FUNCTION_BLOCK AX_RangeBasedPulse (* Generates a pulse on AX adapter based on distance traveled (Adapter Version) *)
  (* Standard: 61499-2; Description: Copyright (c) 2026 HR Agrartechnik GmbH This program and the accompanying materials are made available under the terms of the Eclipse Public License 2.0 which is available at https://www.eclipse.org/legal/epl-2.0/ SPDX-License-Identifier: EPL-2.0 *)
  (* Version 1.0, 2026-04-19, Franz Höpfinger, HR Agrartechnik GmbH, initial API and implementation *)
  PACKAGE logiBUS::signalprocessing::distance;
  IMPORT eclipse4diac::core::TypeHash;
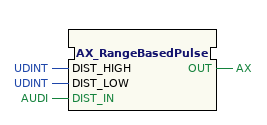
  VAR_INPUT
    DIST_HIGH : UDINT := 5000; (* Distance for HIGH pulse (mm) *)
    DIST_LOW : UDINT := 5000; (* Distance for LOW pulse (mm) *)
  END_VAR
  SOCKETS
    DIST_IN : adapter::types::unidirectional::AUDI; (* Input Distance Adapter *)
  END_SOCKETS
  PLUGS
    OUT : adapter::types::unidirectional::AX; (* Pulse Output Adapter *)
  END_PLUGS
  VAR
    LastDist : UDINT; (* Last distance value when state changed *)
    FirstRun : BOOL := TRUE; (* Initial run flag *)
    LastState : BOOL; (* Last state of Q *)
  END_VAR
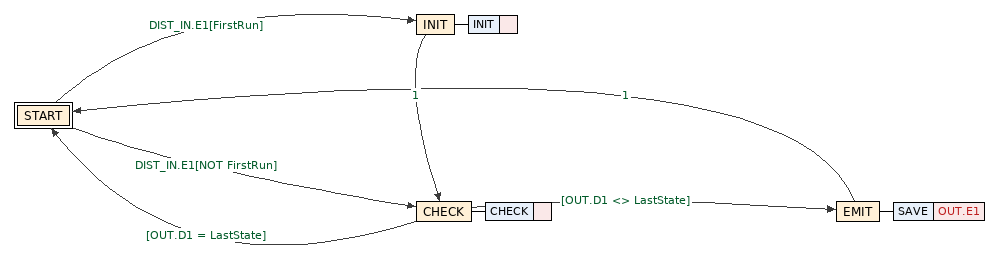
  EC_STATES
    START; (* Initial State *)
    INIT : INIT; (* Initialize base distance *)
    CHECK : CHECK; (* Evaluate distance *)
    EMIT : SAVE -> OUT.E1; (* Fire state change *)
  END_STATES
  EC_TRANSITIONS
    START TO INIT := DIST_IN.E1[FirstRun];
    INIT TO CHECK := 1;
    START TO CHECK := DIST_IN.E1[NOT FirstRun];
    CHECK TO EMIT := [OUT.D1 <> LastState];
    CHECK TO START := [OUT.D1 = LastState];
    EMIT TO START := 1;
  END_TRANSITIONS
  ALGORITHM INIT IN ST:
LastDist := DIST_IN.D1;
OUT.D1 := BOOL#FALSE;
LastState := BOOL#FALSE;
FirstRun := BOOL#FALSE;
  END_ALGORITHM
  ALGORITHM CHECK IN ST:
IF (LastState = BOOL#FALSE) THEN
  IF (DIST_IN.D1 >= (LastDist + DIST_LOW)) THEN
    OUT.D1 := BOOL#TRUE;
    LastDist := DIST_IN.D1;
  END_IF;
ELSE
  IF (DIST_IN.D1 >= (LastDist + DIST_HIGH)) THEN
    OUT.D1 := BOOL#FALSE;
    LastDist := DIST_IN.D1;
  END_IF;
END_IF;
  END_ALGORITHM
  ALGORITHM SAVE IN ST:
LastState := OUT.D1;
  END_ALGORITHM
END_FUNCTION_BLOCK
